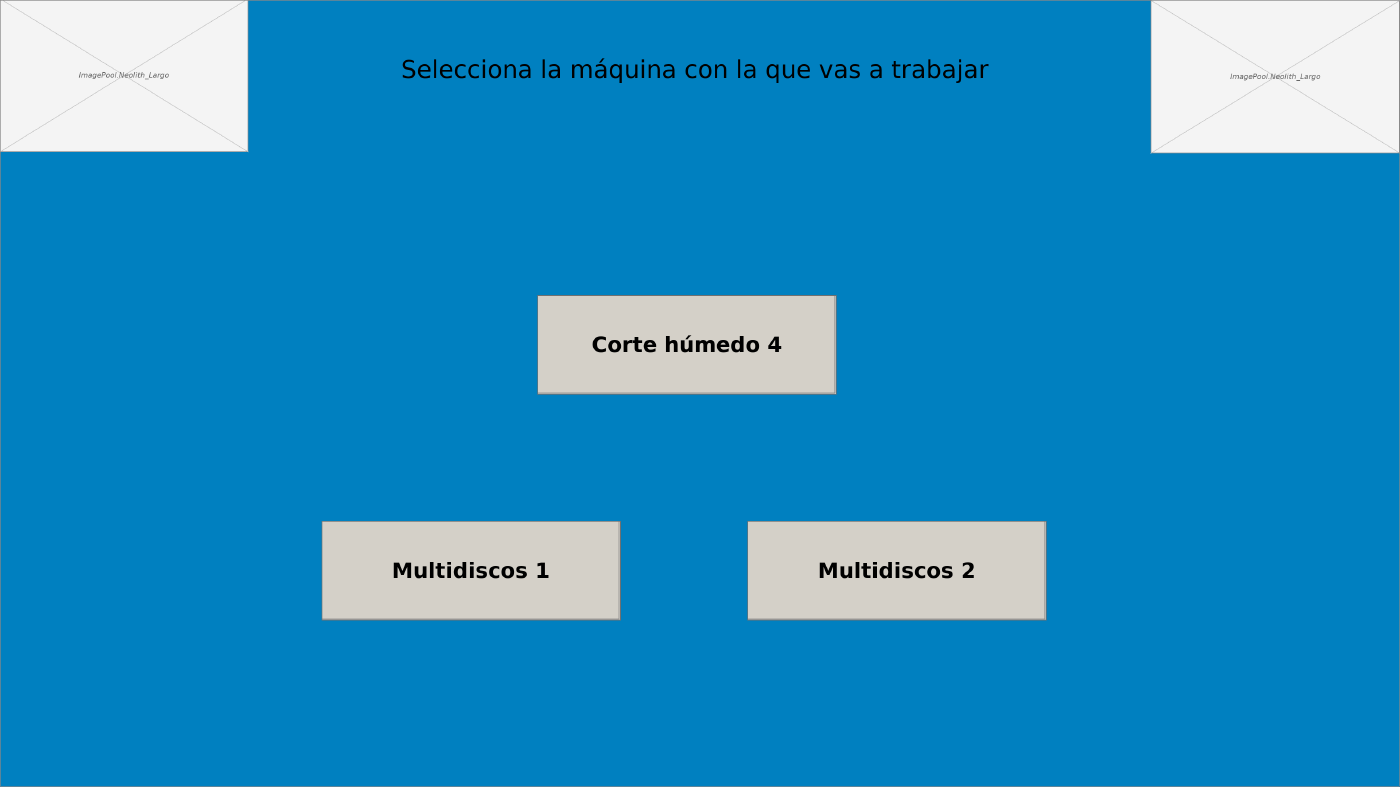
VISUALIZATION Home_Sel_Maq  // 1920x1080
    Label (335,21 1236x148), "Selecciona la máquina con la que vas a trabajar"
    Image (1578,0 342x210), image: ImagePool.Neolith_Largo
    Image (0,-2 340x210), image: ImagePool.Neolith_Largo
    Button (737,405 410x136), "Corte húmedo 4"
        OnMouseUp: change screen: Home_CortH4
    Button (441,715 410x136), "Multidiscos 1"
        OnMouseUp: change screen: Home_Multidis1
    Button (1025,715 410x136), "Multidiscos 2"
        OnMouseDown: change screen: Home_Multidis2
END_VISUALIZATION

(* stored: Version 1.1.0.1, ProductVersion 3.1.4024.12
   Visu Home_Sel_Maq: Id {5257e64c-3155-462c-b35e-deb33ee21df1} *)
